TYPE ST_AXIS_VELOCITY :
STRUCT
END_STRUCT
END_TYPE

(* stored: Version 1.1.0.1, ProductVersion 3.1.4024.11
   DUT ST_AXIS_VELOCITY: Id {e91163e7-f329-462a-adb0-c35f70d24efd} *)
